{attribute 'pack_mode' := '1'}
TYPE IOStatus EXTENDS OutgoingMessage :
STRUCT
	digitalInputs: DINT;  (* Bit mask of current states. *)
	digitalOutputs: DINT; (* Bit mask of current states. *)
	analogInputs: ARRAY [0..CT.ANALOG_ARRAY_SIZE-1] OF LREAL; (* Current analog readings. *)
END_STRUCT
END_TYPE

(* stored: Version 1.1.0.1, ProductVersion 3.1.4022.12
   DUT IOStatus: Id {5fedbb2e-ef0a-458b-9744-96f501654a06} *)
